{attribute 'TcGenerated'}
// This function has been automatically generated from the project information.
VAR_GLOBAL CONSTANT
	{attribute 'const_non_replaced'}
	{attribute 'linkalways'}
	stLibVersion_Unittest : ST_LibVersion := (iMajor := 0, iMinor := 1, iBuild := 0, iRevision := 0, sVersion := '0.1');
END_VAR

(* stored: Version 1.1.0.1, ProductVersion 3.1.4022.9
   GVL Global_Version: Id {1e1ad4cd-5591-4a8a-8e2a-2982e25c4685} *)
